FUNCTION_BLOCK scaleValue
VAR_INPUT
	rInputPercent:REAL;
	rMaxValue:REAL;

END_VAR
VAR_OUTPUT
	
	iScaled:INT;
END_VAR
VAR
END_VAR

iScaled:=REAL_TO_INT(rInputPercent*rMaxValue/100);

END_FUNCTION_BLOCK

(* stored: Version 1.1.0.1, ProductVersion 3.1.4022.12
   POU scaleValue: Id {56cf4de0-2487-416e-a10e-85933b24d267}, SpecialFunc None *)
